FUNCTION_BLOCK CylinderOrchestrator (* Message Exchange example (slide 47): CylMES / CControlTRAS - orchestrates the round trip between the cylinder and the drop sink *)
  (* Standard: 61499-2; Description: Copyright (c) 2026 Meisterschulen am Ostbahnhof This program and the accompanying materials are made available under the terms of the Eclipse Public License 2.0 which is available at https://www.eclipse.org/legal/epl-2.0/ SPDX-License-Identifier: EPL-2.0 *)
  (* Version 1.0, 2026-09-03, Franz Höpfinger, Meisterschulen am Ostbahnhof, SoA implementation in function blocks (IEC 61499 primer course, Module 6, Valeriy Vyatkin, slide 47), CylMES/CControlTRAS role: SRSP (from WorkpieceSensor) and SREQ2 (to DropSinkService) use EVENT_HS_ACK_WSTRING (REQ/CNF only), SREQ1 (to CylinderService) uses full EVENT_HS_WSTRING since it must react to the mid-trip IND. Deliberately omits the slide's TokenRing (MTXIN/MTXOUT) interlock and the constant-TRUE Enable/Permit adapter: this demo has only one controller, so there is nothing to interlock against - see HandshakePattern.md for the full rationale *)
  (* Version 1.1, 2026-09-03, Franz Höpfinger, Meisterschulen am Ostbahnhof, PR #160 review feedback (coderabbitai): CylinderService fires SREQ1.IND twice per trip (RSP_CYL_STARTED, then RSP_CYL_END_POS) but Initialized->REQUEST_DROP reacted to either, requesting the drop prematurely on the started indication. Fixed by gating the transition on SREQ1.INDD = MessageExchangeConst::RSP_CYL_END_POS *)
  PACKAGE Meins::DesingPatterns::HandshakePattern;
  IMPORT Meins::DesingPatterns::HandshakePattern::const::MessageExchangeConst;
  (* Documentation:
  Cylinder orchestrator (CylMES, type CControlTRAS on the slide) in the "SoA implementation in function blocks" diagram (IEC 61499 primer course, Module 6, Valeriy Vyatkin, slide 47) - one of the four function blocks in the CylH message-exchange example (slides 42-46 for the message sequence chart this reconstructs).
   Three adapter connections, exactly as on the slide:
    - SRSP (Socket, EVENT_HS_ACK_WSTRING) towards WorkpieceSensor - receives the trip request, answers once the whole round trip is done.
   - SREQ1 (Plug, full EVENT_HS_WSTRING) towards CylinderService - forwards the trip request; reacts to the mid-trip IND (cylinder reached the end position) by requesting the drop, then answers with RSP once the sink has acknowledged it, letting the cylinder retract.
   - SREQ2 (Plug, EVENT_HS_ACK_WSTRING) towards DropSinkService - requests the drop, waits for its acknowledgement.
    Deliberately omitted vs. the slide: the TokenRing adapter (MTXIN/MTXOUT) for mutual-exclusion interlocking between multiple cylinder controllers, and the constant-TRUE Enable/Permit adapter gating execution. Both exist on the slide for a multi-controller deployment; this demo has exactly one CylinderOrchestrator instance, so there is nothing to interlock against and no reason to gate a permit that is always TRUE. See TokenRingPattern.md for the TokenRing adapter itself, already implemented separately in this repository.
   See HandshakePattern.md in this folder, section "Die Quelle der 'push,100'-Notation", for the full write-up and the other three function blocks of this example (WorkpieceSensor, DropSinkService, CylinderService).
  *)
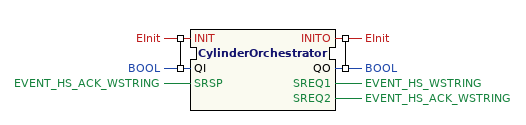
  EVENT_INPUT
    INIT : EInit WITH QI; (* Initialization Request *)
  END_EVENT
  EVENT_OUTPUT
    INITO : EInit WITH QO; (* Initialization Confirm *)
  END_EVENT
  VAR_INPUT
    QI : BOOL; (* Input event qualifier *)
  END_VAR
  VAR_OUTPUT
    QO : BOOL; (* Output event qualifier *)
  END_VAR
  SOCKETS
    SRSP : adapter::types::bidirectional::Handshake::EVENT_HS_ACK_WSTRING; (* Service socket towards WorkpieceSensor: receives the trip REQ (+REQD), answers with CNF (+CNFD) once the whole trip is done *)
  END_SOCKETS
  PLUGS
    SREQ1 : adapter::types::bidirectional::Handshake::EVENT_HS_WSTRING; (* Service plug towards CylinderService: full REQ/CNF/IND/RSP - reacts to the mid-trip IND (reached end position) *)
    SREQ2 : adapter::types::bidirectional::Handshake::EVENT_HS_ACK_WSTRING; (* Service plug towards DropSinkService: REQ/CNF only *)
  END_PLUGS
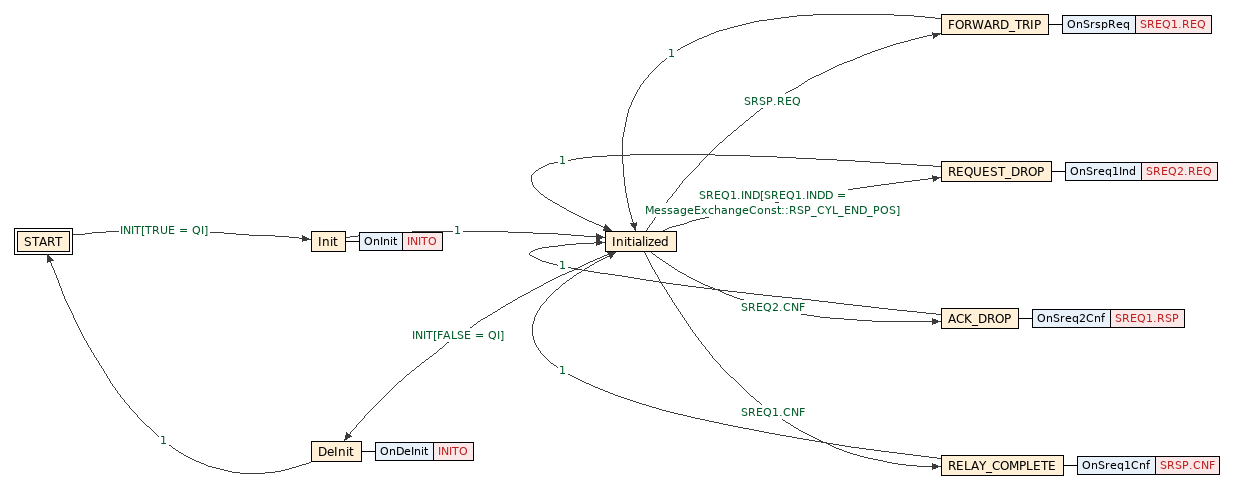
  EC_STATES
    START; (* Uninitialized *)
    Init : OnInit -> INITO; (* Initialization *)
    Initialized; (* Idle, ready to react to any of the three adapters *)
    DeInit : OnDeInit -> INITO; (* De-initialization *)
    FORWARD_TRIP : OnSrspReq -> SREQ1.REQ; (* WorkpieceSensor requested a trip: forward it to the cylinder *)
    REQUEST_DROP : OnSreq1Ind -> SREQ2.REQ; (* Cylinder reached end position: request the sink to accept the workpiece *)
    ACK_DROP : OnSreq2Cnf -> SREQ1.RSP; (* Sink acknowledged the drop: let the cylinder retract *)
    RELAY_COMPLETE : OnSreq1Cnf -> SRSP.CNF; (* Cylinder confirms the trip is complete: relay it to WorkpieceSensor *)
  END_STATES
  EC_TRANSITIONS
    START TO Init := INIT[TRUE = QI];
    Init TO Initialized := 1;
    Initialized TO DeInit := INIT[FALSE = QI];
    DeInit TO START := 1;
    Initialized TO FORWARD_TRIP := SRSP.REQ;
    FORWARD_TRIP TO Initialized := 1;
    Initialized TO REQUEST_DROP := SREQ1.IND[SREQ1.INDD = MessageExchangeConst::RSP_CYL_END_POS];
    REQUEST_DROP TO Initialized := 1;
    Initialized TO ACK_DROP := SREQ2.CNF;
    ACK_DROP TO Initialized := 1;
    Initialized TO RELAY_COMPLETE := SREQ1.CNF;
    RELAY_COMPLETE TO Initialized := 1;
  END_TRANSITIONS
  ALGORITHM OnInit IN ST: (* Initialize *)
QO := QI;
  END_ALGORITHM
  ALGORITHM OnDeInit IN ST: (* De-initialize *)
QO := FALSE;
  END_ALGORITHM
  ALGORITHM OnSrspReq IN ST: (* Pass the trip request through to the cylinder unchanged *)
SREQ1.REQD := SRSP.REQD;
  END_ALGORITHM
  ALGORITHM OnSreq1Ind IN ST: (* Cylinder reported reaching the end position: request the drop *)
SREQ2.REQD := MessageExchangeConst::REQ_DROP;
  END_ALGORITHM
  ALGORITHM OnSreq2Cnf IN ST: (* Sink acknowledged the drop: tell the cylinder it may retract *)
SREQ1.RSPD := MessageExchangeConst::RSP_ACK;
  END_ALGORITHM
  ALGORITHM OnSreq1Cnf IN ST: (* Trip fully complete: relay the confirmation upward *)
SRSP.CNFD := SREQ1.CNFD;
  END_ALGORITHM
END_FUNCTION_BLOCK
